{attribute 'linkalways'} 
{attribute 'no_explicit_call' := 'This FB is a CLASS and must be accessed using methods or properties'}
{attribute 'enable_dynamic_creation'}
FUNCTION_BLOCK FINAL MUL_USINT EXTENDS Node
VAR
	in1 : _USINT(0);
	in2 : _USINT(0);
	out : _USINT(0);
END_VAR

METHOD PUBLIC Clone : I_Node
VAR
	pNode : POINTER TO MUL_USINT;
END_VAR
pNode := __NEW(MUL_USINT);
Clone := pNode^;
END_METHOD

METHOD FB_init : BOOL
VAR_INPUT
	bInitRetains : BOOL; // if TRUE, the retain variables are initialized (warm start / cold start)
	bInCopyCode : BOOL;  // if TRUE, the instance afterwards gets moved into the copy code (online change)
END_VAR
AddInput('in1',THIS^.in1);
AddInput('in2',THIS^.in2);
AddOutput('out', THIS^.out);
END_METHOD

METHOD PROTECTED OnExecute
VAR
END_VAR
out.Value := in1.Value * in2.Value;
END_METHOD

END_FUNCTION_BLOCK

(* stored: Version 1.1.0.1, ProductVersion 3.1.4024.15
   POU MUL_USINT: Id {db348e7c-a834-441b-9d6d-d677638284d9}, SpecialFunc None
   Folder Constructor: Id {dbb4e104-fc24-47c9-89c6-f27de74ebc4c}
   Method Clone: Id {8616e1ae-5775-4fa1-8308-9c81743e6d4e}
   Method FB_init: Id {175af7ca-5aeb-4f06-8044-501b6044ee76}
   Method OnExecute: Id {a960114a-3a78-4e53-b7ca-3ad77a462236} *)
